FUNCTION Function (* Function with empty body *)
  (* Standard: 61499-1 *)
  (* Version 1.0, 2023-06-29, mjobst *)
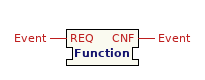
  EVENT_INPUT
    REQ;
  END_EVENT
  EVENT_OUTPUT
    CNF;
  END_EVENT
END_FUNCTION
